# B&R Automation Studio project acopos6d_issues (part 5)

#### FastLib.fun - Exported functions and function blocks
```iecst
FUNCTION_BLOCK fdStationQueueControl
	VAR_INPUT
		Enable : BOOL;
		ReleaseShuttles : BOOL;
		ShuttleList : ARRAY[0..fdSTATION_SHUTTLE_LAST_INDEX] OF MpTrafficShuttleInfoType;
		ShuttleCapacity : UINT; (*Count how many shuttles process station can handle*)
		pStation : REFERENCE TO MpTrafficStationControl;
	END_VAR
	VAR_OUTPUT
		ShuttleReleaseDone : BOOL;
		ShuttleReleaseAborted : BOOL;
		ReleaseShuttle : BOOL;
		NumOccypyingShuttles : UINT;
	END_VAR
	VAR
		state : DINT;
		lastState : DINT;
		loop : DINT;
		index : DINT;
		shuttleFound : BOOL;
		shuttleIDToRelease : UINT;
		shuttleIDToAutoRelease : UINT;
	END_VAR
END_FUNCTION_BLOCK

FUNCTION_BLOCK fdTiltAround
	VAR_INPUT
		Execute : {REDUND_UNREPLICABLE} BOOL;
		MaxAngle : {REDUND_UNREPLICABLE} REAL;
		Steps : {REDUND_UNREPLICABLE} DINT;
		Velocity : McAcp6DShortAxAxesType;
		Shuttle : REFERENCE TO Mc6DShuttleType;
	END_VAR
	VAR_OUTPUT
		Acknowledge : BOOL;
		Error : BOOL;
	END_VAR
	VAR
		state : DINT;
		step : DINT;
		MoveShortAxis : MC_BR_MoveShortAxis_Acp6D;
	END_VAR
END_FUNCTION_BLOCK

FUNCTION_BLOCK fdWaitUntilAllDone
	VAR_INPUT
		Execute : {REDUND_UNREPLICABLE} BOOL;
		Shuttles : {REDUND_UNREPLICABLE} ARRAY[0..fdMAX_WAIT_SHUTTLE_COUNT] OF Mc6DShuttleType;
	END_VAR
	VAR_OUTPUT
		Done : BOOL;
		Error : BOOL;
		WaitingFor : UINT;
	END_VAR
	VAR
		state : DINT;
		i : DINT;
		ShGetInfo : MC_BR_ShGetInfo_Acp6D;
	END_VAR
END_FUNCTION_BLOCK

FUNCTION_BLOCK fdPulse
	VAR_INPUT
		Execute : {REDUND_UNREPLICABLE} BOOL;
		T_on : {REDUND_UNREPLICABLE} TIME;
		T_off : {REDUND_UNREPLICABLE} TIME;
	END_VAR
	VAR_OUTPUT
		Q : BOOL;
	END_VAR
	VAR
		state : DINT;
		TON_on : TON;
		TON_off : TON;
	END_VAR
END_FUNCTION_BLOCK

FUNCTION_BLOCK fdFindZone
	VAR_INPUT
		Assembly : REFERENCE TO Mc6DAssemblyType; (*The assembly reference establishes the connection between the function block and the assembly.*)
		Execute : BOOL;
		Name : STRING[32];
	END_VAR
	VAR_OUTPUT
		ZoneFound : BOOL;
		ZoneNotFound : BOOL;
		Error : BOOL;
		Zone : Mc6DZoneType; (* Zone reference *)
		ZoneInfo : McAcp6DGetZoneAddInfoType;
	END_VAR
	VAR
		state : DINT;
		i : DINT;
		AsmGetZone : MC_BR_AsmGetZone_Acp6D;
		lastZoneID : UINT;
	END_VAR
END_FUNCTION_BLOCK

FUNCTION_BLOCK fdStation
	VAR_INPUT
		Assembly : REFERENCE TO Mc6DAssemblyType;
		TrafficManager : REFERENCE TO MpTrafficManagerType;
		Station : REFERENCE TO MpTrafficStationType;
		NextStation : REFERENCE TO MpTrafficStationType;
		Enable : BOOL;
		NextState : BOOL;
		JumpToState : UINT;
		Parameters : fdStationParametersType;
		Commands : fdStationCommandsType;
		Operation : fdStationOperationType;
		Loop : DINT;
		StateInfo : STRING[80];
	END_VAR
	VAR_OUTPUT
		State : UINT;
		Active : BOOL;
		NumOccupyingShuttles : UINT;
		CommandDone : BOOL;
		CommandAcknowledge : BOOL;
		CommandError : BOOL;
		ErrorID : DINT;
		ErroredSequenceState : DINT;
		Shuttles : fdStationShuttlesType;
		VirtualShuttle : MpTrafficShuttleInfoType;
		MacroShuttle : MpTrafficShuttleInfoType;
	END_VAR
	VAR
		m_sequence_state : DINT;
		m_control : fdStationMemberControlType;
		m_move : fdStationMemberMoveType;
		m_group : fdStationMemberGroupType;
		m_macro : fdStationMemberMacroType;
		m_zone : fdStationMemberZoneType;
		m_cmd : fdStationMemberCommandType;
		m_status : fdStationMemberStatusType;
		m_var : fdStationMemberVarType;
	END_VAR
END_FUNCTION_BLOCK
(**)

FUNCTION_BLOCK fdMove6DSync
	VAR_INPUT
		Shuttle : REFERENCE TO Mc6DShuttleType;
		Execute : BOOL;
		Home : BOOL;
		Parameters : fdMove6DSyncParametersType;
	END_VAR
	VAR_OUTPUT
		Acknowledge : BOOL;
		Done : BOOL;
		Error : BOOL;
		ErrorID : DINT;
		CurrentPosition : McAcp6DShPositionType;
	END_VAR
	VAR
		state : DINT;
		i : DINT;
		ShGetInfo : MC_BR_ShGetInfo_Acp6D;
		Move6D : MC_BR_Move6D_Acp6D;
		m : fdMove6DSyncMemberType;
	END_VAR
END_FUNCTION_BLOCK

FUNCTION fdCalcTimeToTarget : REAL
	VAR_INPUT
		Distance : REAL;
		MaxVelocity : REAL;
		Acceleration : REAL;
	END_VAR
	VAR
		timeToMaxVelocity : REAL;
		distanceToMaxVelocity : REAL;
		distanceToTarget : REAL;
	END_VAR
END_FUNCTION

FUNCTION fdCalcTargetVelocity : REAL
	VAR_INPUT
		Distance : REAL;
		TimeToTarget : REAL;
		Acceleration : REAL;
	END_VAR
	VAR
		minimumVelocity : REAL;
		discriminant : REAL;
		a : REAL;
		b : REAL;
		c : REAL;
		x1 : REAL;
		x2 : REAL;
	END_VAR
END_FUNCTION
```

#### fdStationQueueControl.st
```iecst
(*  *)
FUNCTION_BLOCK fdStationQueueControl

	IF NOT Enable THEN
		state := 0;
		ReleaseShuttle := FALSE;
		ShuttleReleaseDone := FALSE;
		ShuttleReleaseAborted := FALSE;
	END_IF;

	CASE state OF
		0:
			// -----------------------------------------------------------------
			IF ReleaseShuttles THEN
				IF pStation.Info.NumOccupyingShuttles > 0 THEN
					index := 0;
					state := 100;
				ELSE
					state := 199;
				END_IF;
			ELSIF pStation.Info.NumOccupyingShuttles > ShuttleCapacity THEN
				shuttleIDToAutoRelease := pStation.Info.LastArrivedShuttle.ShuttleID;
				// Station is executing current process and there is no room for more shuttles ->
				// release queuing extra shuttles straight forward
				loop := 0;
				state := 200;
			END_IF;

		100:
			// Manual queue release sequence
			// ----------------------------------------------------------------------------------------------------------------------------------
			// Select the next requested shuttle from the shuttle list
			shuttleFound := FALSE;

			WHILE index <= fdSTATION_SHUTTLE_LAST_INDEX DO
				IF ShuttleList[index].ShuttleID > 0 THEN
					shuttleIDToRelease := ShuttleList[index].ShuttleID;
					shuttleFound := TRUE;
					index := index + 1;
					EXIT;
				END_IF;
				index := index + 1;
			END_WHILE;

			IF shuttleFound THEN
				// Proceed to release next shuttle
				loop := 0;
				state := 110;
			ELSE
				// No more shuttles to release
				state := 199;
			END_IF;
		110:
			// Select shuttle to be released from stations shuttle list
			// -----------------------------------------------------------------
			IF loop > pStation.Info.NumOccupyingShuttles THEN
				// whole list has been checked through and we cant find requested shuttle -> move on
				state := 100;
			ELSIF pStation.SelectedShuttle.ShuttleID = shuttleIDToRelease THEN
				state := 130;
			ELSE
				loop := loop  + 1;
				pStation(SelectNextShuttle := TRUE);
				pStation(SelectNextShuttle := FALSE);
			END_IF;
		130:
			// Release the shuttle
			// -----------------------------------------------------------------
			ReleaseShuttle := TRUE;

			IF pStation.ReleaseDone THEN
				state := 100;
			ELSIF pStation.ReleaseAborted THEN
				state := 300;
			END_IF;
		199:
			// Done
			// -----------------------------------------------------------------
			ShuttleReleaseDone := TRUE;

			IF NOT ReleaseShuttles THEN
				state := 0;
			END_IF;

		200:
			// Automatic queue release sequence
			// ----------------------------------------------------------------------------------------------------------------------------------
			// Select shuttle to be released from stations shuttle list
			// -----------------------------------------------------------------
			IF loop > pStation.Info.NumOccupyingShuttles THEN
				// whole list has been checked through and we cant find requested shuttle -> move on
				state := 0;
			ELSIF pStation.SelectedShuttle.ShuttleID = shuttleIDToAutoRelease THEN
				state := 210;
			ELSE
				loop := loop  + 1;
				pStation(SelectNextShuttle := TRUE);
				pStation(SelectNextShuttle := FALSE);
			END_IF;
		210:
			// Release the queuing shuttle
			// -----------------------------------------------------------------
			ReleaseShuttle := TRUE;

			IF pStation.ReleaseDone THEN
				state := 0;
			ELSIF pStation.ReleaseAborted THEN
				state := 300;
			END_IF;

		300:
			// Error
			// -----------------------------------------------------------------
			ShuttleReleaseAborted := TRUE;

	END_CASE;

	IF state <> lastState THEN
		lastState := state;
		ReleaseShuttle := FALSE;
		ShuttleReleaseDone := FALSE;
		ShuttleReleaseAborted := FALSE;
	END_IF;

	NumOccypyingShuttles := pStation.Info.NumOccupyingShuttles;

END_FUNCTION_BLOCK
```

#### fdTiltAround.st
```iecst
(*  *)
FUNCTION_BLOCK fdTiltAround

	IF NOT Execute THEN
		MoveShortAxis.Execute := FALSE;
		step := 0;
		state := 0;
	END_IF;

	CASE state OF
		0:
			IF Execute THEN
				state := 10;
			END_IF;
		10:
			IF step > Steps THEN
				state := 100;
			ELSE
				MoveShortAxis.Parameters.Position.Rx := MaxAngle * SIN((2 * brmPI / Steps) * step);
				MoveShortAxis.Parameters.Position.Ry := MaxAngle * COS((2 * brmPI / Steps) * step);
				MoveShortAxis.Parameters.Position.Rz := 0;
				MoveShortAxis.Parameters.Position.Z := 0.004;
				state := 20;
			END_IF;
		20:
			MoveShortAxis.Execute := TRUE;

			IF MoveShortAxis.Acknowledge THEN
				MoveShortAxis.Execute := FALSE;
				step := step + 1;
				state := 10;
			END_IF;
		100:
//			MoveShortAxis.Parameters.Position.Rx := 0;
//			MoveShortAxis.Parameters.Position.Ry := 0;
//			MoveShortAxis.Parameters.Position.Rz := 0;
//			MoveShortAxis.Parameters.Position.Z := 0.001;
//			MoveShortAxis.Execute := TRUE;
//
//			IF MoveShortAxis.Done OR MoveShortAxis.Acknowledge THEN
//				MoveShortAxis.Execute := FALSE;
//				step := step + 1;
//				state := 101;
//			END_IF;

			IF NOT Execute THEN
				state := 0;
			END_IF;
	END_CASE;

	MoveShortAxis.Shuttle := ADR(Shuttle);
	MoveShortAxis.Parameters.Mode :=  mcACP6D_MOVE_ABSOLUTE;
	MoveShortAxis.Parameters.Velocity := Velocity;
	MoveShortAxis();

	Acknowledge := (state = 100);
	Error := MoveShortAxis.Error;

END_FUNCTION_BLOCK
```

#### fdWaitUntilIdle.st
```iecst
(*  *)
FUNCTION_BLOCK fdWaitUntilAllDone

	IF NOT Execute THEN
		state := 0;
		i := 0;
		ShGetInfo.Execute := FALSE;
		WaitingFor := 0;
	END_IF;

	CASE state OF
		0:
			IF Execute THEN
				state := 10;
			END_IF;
		10:
			IF i > fdMAX_STATION_SHUTTLE_COUNT THEN
				state := 100;
			ELSE
				IF Shuttles[i].controlif = 0 THEN
					// Not a valid shuttle reference. Move to next item in the list
					i := i + 1;
				ELSE
					state := 20;
				END_IF;
			END_IF;
		20:
			ShGetInfo.Execute := TRUE;

			IF ShGetInfo.Done THEN
				WaitingFor := ShGetInfo.ShuttleInfo.ShuttleID;

				IF (ShGetInfo.ShuttleInfo.State =  mcACP6D_SH_STATE_IDLING) AND (ShGetInfo.ShuttleInfo.MotionBuffer.NumberOfCommands = 0) THEN
					i := i + 1;
					state := 10;
				END_IF;
				ShGetInfo.Execute := FALSE;

			ELSIF ShGetInfo.Error THEN
				ShGetInfo.Execute := FALSE;
				state := 101;
			END_IF;
		100:
			IF NOT Execute THEN
				state := 0;
			END_IF;
	END_CASE;

	ShGetInfo.Shuttle := ADR(Shuttles[i]);
	ShGetInfo();

	Done := (state = 100);
	Error := ShGetInfo.Error;

END_FUNCTION_BLOCK
```

#### fdPulse.st
```iecst
(*  *)
FUNCTION_BLOCK fdPulse

	IF NOT Execute THEN
		state := 0;
	END_IF;

	CASE state OF
		0:
			IF Execute THEN
				state := 10;
			END_IF;
		10:
			IF TON_on.Q THEN
	  			state := 20;
			END_IF;
		20:
			IF TON_off.Q THEN
				state := 10;
			END_IF;
		100:
			IF NOT Execute THEN
				state := 0;
			END_IF;
	END_CASE;

	TON_on.IN := (state = 10);
	TON_on.PT := T_on;
	TON_on();

	TON_off.IN := (state = 20);
	TON_off.PT := T_off;
	TON_off();

	Q := (state = 10);

END_FUNCTION_BLOCK
```

#### fdFindZone.st
```iecst
(*  *)
FUNCTION_BLOCK fdFindZone

	IF NOT Execute THEN
		state := 0;
		i := 0;
		AsmGetZone.Enable := FALSE;
		ZoneFound := FALSE;
		ZoneNotFound := FALSE;
		Error := FALSE;
		brsmemset(ADR(ZoneInfo), 0, SIZEOF(ZoneInfo));
		brsmemset(ADR(Zone), 0, SIZEOF(Zone));
	END_IF;

	CASE state OF
		0:
			// --------------------------------------------
			IF Execute THEN
				state := 10;
			END_IF;
		10:
			// --------------------------------------------
			AsmGetZone.Enable := TRUE;
			IF AsmGetZone.Valid THEN
				IF AsmGetZone.TotalCount = 0 THEN
					state := 101;
				ELSE
					state := 20;
				END_IF;
			END_IF;
		20:
			// --------------------------------------------
			lastZoneID := AsmGetZone.AdditionalInfo.ZoneID;

			IF brsmemcmp(ADR(AsmGetZone.AdditionalInfo.Name), ADR(Name), SIZEOF(Name)) = 0 THEN
				// Names match -> found
				Zone := AsmGetZone.Zone;
				ZoneInfo := AsmGetZone.AdditionalInfo;
				state := 100;
			ELSE
				IF AsmGetZone.RemainingCount = 0 THEN
					state := 101;
				ELSE
					state := 30;
				END_IF;
			END_IF;
		30:
			// --------------------------------------------
			IF AsmGetZone.AdditionalInfo.ZoneID <> lastZoneID THEN
				state := 20;
			END_IF;

		100:
			// --------------------------------------------
			ZoneFound := TRUE;
		101:
			// --------------------------------------------
			ZoneNotFound := TRUE;
		102:
			// --------------------------------------------
			Error := TRUE;
	END_CASE;

	AsmGetZone.Assembly := ADR(Assembly);
	AsmGetZone.Next := (state = 30);
	AsmGetZone();

END_FUNCTION_BLOCK
```

#### fdMove6DSync.st
```iecst
//
FUNCTION fdCalcTimeToTarget

	// v = a * t -> t = v / a
	timeToMaxVelocity := MaxVelocity / Acceleration;

	// Displacement: s = v_0 * t + 0.5 * at^2 -> s = 0.5 * at^2
	distanceToMaxVelocity := 0.5 * Acceleration * brmpow(timeToMaxVelocity, 2);

	// Displacement: s = v_0 * t + 0.5 * at^2 -> t = sqrt((2s)/a)
	IF distanceToMaxVelocity > Distance THEN
		// Case where we never hit the target velocity
		fdCalcTimeToTarget := SQRT(2 * Distance / Acceleration);
	ELSE
		// Case where we reach target velocity
		distanceToTarget := Distance - distanceToMaxVelocity;

		fdCalcTimeToTarget := SQRT(2 * distanceToMaxVelocity / Acceleration) + distanceToTarget / MaxVelocity;
	END_IF;

END_FUNCTION

//
FUNCTION fdCalcTargetVelocity

	// This seems to be rougly minimum velocity 6D system can do
	minimumVelocity := 0.0001;

	IF Distance < 0.001 THEN
		fdCalcTargetVelocity := minimumVelocity;
	END_IF;

	// Move consists of two parts, 1st is acceleration to end velocity and 2nd is constant velocity part
	// We know following:
	// TimeToTarget = t1 + t2
	// TargetVelocity = Acceleration * t1
	// s2 = TargetVelocity * t2
	// Distance = s1 + s2
	// s1 = 0.5 * Acceleration * t1^2

	// Solve with quadratic equation
	// x = (-b +- SQRT((b^2)-4ac))/2a
	// discriminant = b*b - 4*a*c;
	a := 0.5;
	b := -1 * TimeToTarget * Acceleration;
	c := Acceleration * Distance;

	// Solve discriminant for the equation
	discriminant := b * b - 4 * a * c;

	IF (discriminant > 0) THEN
		// Two real and distinct roots
		x1 := (-1 * b + SQRT(discriminant)) / (2*a);
		x2 := (-1 * b - SQRT(discriminant)) / (2*a);

		IF x1 >= 0 AND x2 >= 0 THEN
			fdCalcTargetVelocity := MIN(x1, x2);
		ELSIF x1 > 0 THEN
			fdCalcTargetVelocity := x1;
		ELSIF x2 > 0 THEN
			fdCalcTargetVelocity := x2;
		ELSE
			// Both are negative -> impossible situation as velocity cant be negative in this case
			fdCalcTargetVelocity := 0;
		END_IF;

	ELSIF (discriminant = 0) THEN
		// One real root (repeated)
		fdCalcTargetVelocity := -1 * b / (2*a);
	ELSE
		// No real solution -> set to zero so it errors out as this is impossible request
		fdCalcTargetVelocity := 0;
	END_IF

	//fdCalcTargetVelocity := MAX(MinimumVelocity, fdCalcTargetVelocity);

END_FUNCTION

(*  *)
FUNCTION_BLOCK fdMove6DSync

	CASE state OF
		0:
			// --------------------------------------------
			ShGetInfo.Execute := FALSE;
			Move6D.Execute := FALSE;
			ErrorID := 0;
			m.PositionUpdatePending := FALSE;

			IF Execute THEN
				state := 100;
			ELSIF Home THEN
				state := 200;
			END_IF;

		100:
			// Calculate target velocities for all axis
			// --------------------------------------------
			// Calculate distance each axis needs to travel
			m.DistanceToTarget.InPlane := SQRT(brmpow(Parameters.Position.X - CurrentPosition.X, 2) + brmpow(Parameters.Position.Y - CurrentPosition.Y, 2));
			m.DistanceToTarget.Z := ABS(Parameters.Position.Z - CurrentPosition.Z);
			m.DistanceToTarget.Rx := ABS(Parameters.Position.Rx - CurrentPosition.Rx);
			m.DistanceToTarget.Ry := ABS(Parameters.Position.Ry - CurrentPosition.Ry);
			m.DistanceToTarget.Rz := ABS(Parameters.Position.Rz - CurrentPosition.Rz);

			// Calculate which axis takes longest to reach its target from current position
			m.TimeToTarget.InPlane := fdCalcTimeToTarget(m.DistanceToTarget.InPlane, Parameters.Velocity.InPlane, Parameters.Acceleration.InPlane);
			m.TimeToTarget.Z := fdCalcTimeToTarget(m.DistanceToTarget.Z, Parameters.Velocity.Z, Parameters.Acceleration.Z);
			m.TimeToTarget.Rx := fdCalcTimeToTarget(m.DistanceToTarget.Rx, Parameters.Velocity.Rx, Parameters.Acceleration.Rx);
			m.TimeToTarget.Ry := fdCalcTimeToTarget(m.DistanceToTarget.Ry, Parameters.Velocity.Ry, Parameters.Acceleration.Ry);
			m.TimeToTarget.Rz := fdCalcTimeToTarget(m.DistanceToTarget.Rz, Parameters.Velocity.Rz, Parameters.Acceleration.Rz);

			// The axis that takes the longest to reach the target
			m.LongestTimeToTarget := MAX(m.TimeToTarget.InPlane, m.TimeToTarget.Z, m.TimeToTarget.Rx, m.TimeToTarget.Ry, m.TimeToTarget.Rz);

			m.TargetVelocity.InPlane := fdCalcTargetVelocity(m.DistanceToTarget.InPlane, m.LongestTimeToTarget, Parameters.Acceleration.InPlane);
			m.TargetVelocity.Z := fdCalcTargetVelocity(m.DistanceToTarget.Z, m.LongestTimeToTarget, Parameters.Acceleration.Z);
			m.TargetVelocity.Rx := fdCalcTargetVelocity(m.DistanceToTarget.Rx, m.LongestTimeToTarget, Parameters.Acceleration.Rx);
			m.TargetVelocity.Ry := fdCalcTargetVelocity(m.DistanceToTarget.Ry, m.LongestTimeToTarget, Parameters.Acceleration.Ry);
			m.TargetVelocity.Rz := fdCalcTargetVelocity(m.DistanceToTarget.Rz, m.LongestTimeToTarget, Parameters.Acceleration.Rz);

			state := 101;
		101:
			// Execute the move
			// -------------------------------------------
			Move6D.Parameters.InPlane.Acceleration := Parameters.Acceleration.InPlane;
			Move6D.Parameters.InPlane.Velocity := m.TargetVelocity.InPlane;
			Move6D.Parameters.InPlane.Position.X := Parameters.Position.X;
			Move6D.Parameters.InPlane.Position.Y := Parameters.Position.Y;

			Move6D.Parameters.ShortAxis.Velocity.Z := m.TargetVelocity.Z;
			Move6D.Parameters.ShortAxis.Velocity.Rx := m.TargetVelocity.Rx;
			Move6D.Parameters.ShortAxis.Velocity.Ry := m.TargetVelocity.Ry;
			Move6D.Parameters.ShortAxis.Velocity.Rz := m.TargetVelocity.Rz;
			Move6D.Parameters.ShortAxis.Position.Z := Parameters.Position.Z;
			Move6D.Parameters.ShortAxis.Position.Rx := Parameters.Position.Rx;
			Move6D.Parameters.ShortAxis.Position.Ry := Parameters.Position.Ry;
			Move6D.Parameters.ShortAxis.Position.Rz := Parameters.Position.Rz;
			Move6D.Execute := TRUE;

			IF Move6D.Done OR Move6D.Acknowledge THEN
	  			m.PositionUpdatePending := TRUE;
			END_IF;

			IF NOT Execute THEN
				IF m.PositionUpdatePending THEN
					m.PositionUpdatePending := FALSE;
	  				CurrentPosition := Parameters.Position;
				END_IF;
				Move6D.Execute := FALSE;
				state := 0;
			END_IF;

		200:
			// Home shuttle by reading its current location
			// --------------------------------------------
			ShGetInfo.Execute := TRUE;

			IF NOT Home THEN
				ShGetInfo.Execute := FALSE;
				state := 0;
			ELSIF ShGetInfo.Done THEN
				CurrentPosition := ShGetInfo.ShuttleInfo.Position;
			ELSIF ShGetInfo.Error THEN
				ErrorID := ShGetInfo.ErrorID;
			END_IF;
	END_CASE;

	// Functions
	// --------------------------------------------
	ShGetInfo.Shuttle := ADR(Shuttle);
	ShGetInfo();

	Move6D.Shuttle := ADR(Shuttle);
	Move6D();

	// --------------------------------------------
	Done := Move6D.Done OR ShGetInfo.Done;
	Acknowledge := Move6D.Acknowledge;
	Error := Move6D.Error OR ShGetInfo.Done;

END_FUNCTION_BLOCK
```

#### fdStation.st
```iecst
(* *)
FUNCTION_BLOCK fdStation

	// Station enable control
	// ----------------------------------------------------------------------------------------
	m_control.Enable_EdgeNegative(CLK := Enable);

	IF m_control.Enable_EdgeNegative.Q THEN
		IF Active THEN
			// Jump to
	  		m_sequence_state := 90;
		ELSE
			m_sequence_state := 0;
		END_IF;
	END_IF;

	// External state control
	// ----------------------------------------------------------------------------------------
	IF Active THEN
		IF NextState THEN
			State := State + 1;
			m_var.StateChanged := TRUE;
		ELSIF JumpToState <> State THEN
			State := JumpToState;
			m_var.StateChanged := TRUE;
		END_IF;

		IF m_var.StateChanged THEN
			m_var.StateChanged := FALSE;
			NextState := FALSE;
			JumpToState := State;;
			brsmemset(ADR(Commands), 0, SIZEOF(Commands));
			JumpToState := State;;
		END_IF;
	END_IF;

	// Check if all commands are reset
	// -----------------------------------------------------------------
	m_var.NoCommandActive := (brsmemcmp(ADR(m_var.NoCommands), ADR(Commands), SIZEOF(Commands)) = 0);

	// Station command sequence
	// -----------------------------------------------------------------
	CASE m_sequence_state OF
		0:
			StateInfo := 'Station disabled';
			// -----------------------------------------------------------------
			Active := FALSE;
			State := 0;
			NextState := FALSE;
			JumpToState := 0;
			Loop := 0;
			brsmemset(ADR(Commands), 0, SIZEOF(Commands));
			brsmemset(ADR(Operation), 0, SIZEOF(Operation));
			brsmemset(ADR(m_var), 0, SIZEOF(m_var));
			brsmemset(ADR(m_cmd), 0, SIZEOF(m_cmd));
			brsmemset(ADR(m_status), 0, SIZEOF(m_status));

			IF Enable THEN
	  			m_sequence_state := m_sequence_state + 1;
			END_IF;
		1:
			StateInfo := 'Wait for station to be active and open';
			// -----------------------------------------------------------------
			IF m_control.StationControl.Active AND m_control.StationControl.State = mpTRAFFIC_ST_ON_OPEN THEN
				m_sequence_state := m_sequence_state + 1;
			END_IF
		2:
			StateInfo := 'Create shuttle group';
			// -----------------------------------------------------------------
			m_cmd.GroupCreate := TRUE;
			IF m_group.Create.Done THEN
				m_var.ShuttleGroup := m_group.Create.ShuttleGroup;
				m_sequence_state := 10;
			ELSIF m_group.Create.Error THEN
				m_status.ErrorID := m_group.Create.ErrorID;
			END_IF;
		10:
			StateInfo := 'Check if virtual shuttle exists';
			// -----------------------------------------------------------------
			IF NOT Parameters.CreateVirtualShuttle THEN
				// Virtual shuttle not needed in this station -> move on
				brsmemset(ADR(VirtualShuttle), 0, SIZEOF(VirtualShuttle));
				m_sequence_state := 20;
			ELSE
				IF VirtualShuttle.Shuttle6D.controlif = 0 THEN
					// Virtual shuttle does not exist -> create new one
					m_sequence_state := m_sequence_state + 1;
				ELSE
					// Virtual shuttle already exists in this station -> read its information
					m_sequence_state := 12;
				END_IF;
			END_IF;
		11:
			StateInfo := 'Create virtual shuttle';
			// -----------------------------------------------------------------
			m_cmd.VirtualShuttleCreate := TRUE;

			IF m_control.VirtualShuttleCreate.Done THEN
				VirtualShuttle.Shuttle6D := m_control.VirtualShuttleCreate.VirtualShuttle;
				m_sequence_state := m_sequence_state + 1;
			ELSIF m_control.VirtualShuttleCreate.Error THEN
				m_status.ErrorID := m_control.VirtualShuttleCreate.ErrorID;
			END_IF;
		12:
			StateInfo := 'Read virtual shuttle ID';
			// -----------------------------------------------------------------
			m_control.GetShuttleInfo.Shuttle := ADR(VirtualShuttle.Shuttle6D);
			m_cmd.GetShuttleInfo := TRUE;

			IF m_control.GetShuttleInfo.Done THEN
				VirtualShuttle.ShuttleID := m_control.GetShuttleInfo.ShuttleInfo.ShuttleID;
				m_sequence_state := 20;
			ELSIF m_control.GetShuttleInfo.Error THEN
				m_status.ErrorID := m_control.GetShuttleInfo.ErrorID;
			END_IF;

		20:
			StateInfo := 'Find station zone by name';
			// -----------------------------------------------------------------
			IF brsstrlen(ADR(Parameters.Zone.Name)) = 0 THEN
				m_var.str := DINT_TO_STRING(Parameters.StationNumber);
				Parameters.Zone.Name := CONCAT('Zone', m_var.str);
			END_IF;

			brsmemset(ADR(m_zone.Zone), 0, SIZEOF(m_zone.Zone));
			m_zone.Find.Name := Parameters.Zone.Name;
			m_cmd.ZoneFind := TRUE;

			IF m_zone.Find.ZoneFound THEN
				m_zone.Zone := m_zone.Find.Zone;
				m_sequence_state := 30;
			ELSIF m_zone.Find.ZoneNotFound THEN
				m_sequence_state := m_sequence_state + 1;
			END_IF;
		21:
			StateInfo := 'Create zone';
			// -----------------------------------------------------------------
			m_zone.Create.Parameters.BottomLeft := Parameters.Zone.BottomLeft;
			m_zone.Create.Parameters.TopRight := Parameters.Zone.TopRight;
			m_zone.Create.Parameters.Name := Parameters.Zone.Name;
			m_cmd.ZoneCreate := TRUE;

			IF m_zone.Create.Done THEN
				// Go back one step and rescan the zones to get the zone reference
				m_sequence_state := 20;
			ELSIF m_zone.Create.Error THEN
				m_status.ErrorID := m_zone.Create.ErrorID;
			END_IF;

		30:
			StateInfo := 'Delete old macro if it exists';
			// -----------------------------------------------------------------
			IF brsstrlen(ADR(Parameters.MacroName)) = 0 THEN
				m_var.str := DINT_TO_STRING(Parameters.StationNumber);
				Parameters.MacroName := CONCAT('Macro', m_var.str);
			END_IF;

			m_macro.Delete.Name := Parameters.MacroName;
			m_cmd.MacroDelete := TRUE;

			// Move forward if "macro name not defined" error is received
			IF (m_macro.Delete.Done) OR (m_macro.Delete.Error AND m_macro.Delete.ErrorID = - 1065811714) THEN
				m_sequence_state := m_sequence_state + 1;
			ELSIF m_macro.Delete.Error THEN
				m_status.ErrorID := m_macro.Delete.ErrorID;
			END_IF;
		31:
			StateInfo := 'Create new macro';
			// -----------------------------------------------------------------
			m_macro.Create.Parameters.Name := Parameters.MacroName;
			m_cmd.MacroCreate := TRUE;

			IF m_macro.Create.Done THEN
				m_var.MacroShuttle.Shuttle6D := m_macro.Create.MacroShuttle;
				m_sequence_state := 100;
			ELSIF m_macro.Create.Error THEN
				m_status.ErrorID := m_macro.Create.ErrorID;
			END_IF;

		90:
			StateInfo := 'Deactivating - Clear group';
			// -----------------------------------------------------------------
			m_cmd.GroupClear := TRUE;
			IF m_group.Clear.Done THEN
	  			m_sequence_state := m_sequence_state + 1;
			END_IF;
		91:
			StateInfo := 'Deactivating - Delete group';
			// -----------------------------------------------------------------
			m_cmd.GroupDelete := TRUE;
			IF m_group.Delete.Done THEN
				m_sequence_state := m_sequence_state + 1;
			END_IF;
		92:
			StateInfo := 'Deactivating - Decouple planet system';
			// -----------------------------------------------------------------
			FOR m_var.index := 0 TO fdSTATION_SHUTTLE_LAST_INDEX DO
				m_move.SunPlanet.Parameters.ShuttleList[m_var.index].Shuttle := ADR(m_var.Shuttles.List[m_var.index].Shuttle6D);
			END_FOR;

			m_move.SunPlanet.Parameters.Option := mcACP6D_PLANET_REMOVE_SH;
			m_cmd.Input.SunPlanet.Decouple := TRUE;

			IF m_move.SunPlanet.Done OR (m_move.SunPlanet.ErrorID = -1065795584) THEN
				// Error -1065795584 indicates invalid parameters. A generic issue if shuttles are not currently
				// grouped around sun shuttle. -> just move on
	  			m_sequence_state := m_sequence_state + 1;
			END_IF;
		93:
			StateInfo := 'Deactivating - Delete macro';
			// -----------------------------------------------------------------
			m_cmd.MacroDelete := TRUE;
			IF m_macro.Delete.Done THEN
				m_sequence_state := 99;
			END_IF;
		99:
			StateInfo := 'Deactivating - Deactivation complete';
			// -----------------------------------------------------------------
			m_sequence_state := 0;

		100:
			// Waiting for commands
			// -----------------------------------------------------------------
			Active := TRUE;

			IF Commands.AddShuttle THEN
				m_sequence_state := 110;
			ELSIF Commands.ReleaseAllShuttles THEN
				m_sequence_state := 120;
			ELSIF Commands.MacroRun THEN
				m_sequence_state := 130;
			ELSIF Commands.MacroSave THEN
				m_sequence_state := 140;
			ELSIF Commands.MoveInPlane THEN
				m_sequence_state := 150;
			ELSIF Commands.MoveArc THEN
				m_sequence_state := 160;
			ELSIF Commands.MoveShortAxis THEN
				m_sequence_state := 170;
			ELSIF Commands.Move6D THEN
				m_sequence_state := 180;
			ELSIF Commands.Spin THEN
				m_sequence_state := 190;
			ELSIF Commands.WaitCommandLabel THEN
				m_sequence_state := 200;
			ELSIF Commands.WaitUntilAllDone THEN
				m_sequence_state := 210;
			ELSIF Commands.Group.Couple_CommonCenterPoint THEN
				m_sequence_state := 220;
			ELSIF Commands.Group.Couple_OwnCenterPoint THEN
				m_sequence_state := 221;
			ELSIF Commands.Group.Decouple THEN
				m_sequence_state := 230;
			ELSIF Commands.SunPlanet.Couple THEN
				m_sequence_state := 240;
			ELSIF Commands.SunPlanet.Decouple THEN
				m_sequence_state := 250;
			END_IF;

		110:
			// Add new shuttle to station if there is room for it
			// -----------------------------------------------------------------
			IF m_var.NoCommandActive THEN
				m_sequence_state := 100;
			ELSIF m_var.Shuttles.Count <= fdSTATION_SHUTTLE_LAST_INDEX THEN
				m_var.Shuttles.List[m_var.Shuttles.Count] := m_control.StationControl.Info.LastArrivedShuttle;
				m_var.Shuttles.Count := m_var.Shuttles.Count + 1;
				m_sequence_state := m_sequence_state + 1;
			ELSE
				m_status.CommandError := TRUE;
				m_status.ErrorID := m_sequence_state;
			END_IF;

		111:
			// Clear group before adding ALL shuttles as we cant add one by one
			// -----------------------------------------------------------------
			m_cmd.GroupClear := TRUE;

			m_status.CommandError := m_group.Clear.Error;
			m_status.ErrorID := m_group.Clear.ErrorID;

			IF m_var.NoCommandActive THEN
				m_sequence_state := 100;
			ELSIF m_group.Clear.Done THEN
				m_sequence_state := m_sequence_state + 1;
			END_IF;
		112:
			// Add shuttles to shuttle group
			// -----------------------------------------------------------------
			brsmemset(ADR(m_group.AddShuttle.Parameters.ShuttleList), 0, SIZEOF(m_group.AddShuttle.Parameters.ShuttleList));

			FOR m_var.index := 0 TO m_var.Shuttles.Count - 1 DO
				m_group.AddShuttle.Parameters.ShuttleList[m_var.index].Shuttle := ADR(m_var.Shuttles.List[m_var.index].Shuttle6D);
			END_FOR;

			m_cmd.GroupAddShuttle := TRUE;

			m_status.CommandDone := m_group.AddShuttle.Done;
			m_status.CommandError := m_group.AddShuttle.Error;
			m_status.ErrorID := m_group.AddShuttle.ErrorID;

			IF m_var.NoCommandActive THEN
				m_sequence_state := 100;
			END_IF;

		120:
			// Clear group
			// -----------------------------------------------------------------
			m_cmd.GroupClear := TRUE;

			m_status.CommandError := m_group.Clear.Error;
			m_status.ErrorID := m_group.Clear.ErrorID;

			IF m_var.NoCommandActive THEN
				m_sequence_state := 100;
			ELSIF m_group.Clear.Done THEN
				m_sequence_state := m_sequence_state + 1;
			END_IF;

		121:
			// Release shuttles from station
			// -----------------------------------------------------------------
			m_cmd.Input.ReleaseAllShuttles := TRUE;

			m_status.CommandError := m_control.StationQueueControl.ShuttleReleaseAborted;
			m_status.ErrorID := m_sequence_state;

			IF m_var.NoCommandActive THEN
				m_sequence_state := 100;
			ELSIF m_control.StationQueueControl.ShuttleReleaseDone THEN
				m_sequence_state := m_sequence_state + 1;
			END_IF;

		122:
			// Wait until shuttles have left the station
			// -----------------------------------------------------------------
			m_cmd.ZoneGetBarrierInfo := TRUE;

			m_status.CommandError := m_zone.GetBarrierInfo.Error;
			m_status.ErrorID := m_zone.GetBarrierInfo.ErrorID;

			IF m_var.NoCommandActive THEN
				m_sequence_state := 100;
			ELSIF m_zone.GetBarrierInfo.Done THEN
				m_cmd.ZoneGetBarrierInfo := FALSE;
				IF m_zone.GetBarrierInfo.BarrierInfo.NumberOfShuttles = 0 THEN
					m_var.Shuttles.Count := 0;
					brsmemset(ADR(m_var.Shuttles.List), 0, SIZEOF(m_var.Shuttles.List));
					m_status.CommandDone := TRUE;
				END_IF;
			END_IF;

		130:
			// Run macro command
			// -----------------------------------------------------------------
			m_macro.Run.Name := Parameters.MacroName;
			m_cmd.Input.MacroRun := TRUE;

			m_status.CommandDone := m_macro.Run.Done;
			m_status.CommandAcknowdledge := m_macro.Run.Acknowledge;
			m_status.CommandError := m_macro.Run.Error;
			m_status.ErrorID := m_macro.Run.ErrorID;

			IF m_var.NoCommandActive THEN
				m_sequence_state := 100;
			END_IF;

		140:
			// Save macro command
			// -----------------------------------------------------------------
			m_cmd.Input.MacroSave := TRUE;

			m_status.CommandDone := m_macro.Save.Done;
			m_status.CommandError := m_macro.Save.Error;
			m_status.ErrorID := m_macro.Save.ErrorID;

			IF m_var.NoCommandActive THEN
				m_sequence_state := 100;
			END_IF;

		150:
			// Move in plane command
			// -----------------------------------------------------------------
			m_move.MoveInPlane.Parameters := Operation.MoveInPlane;
			m_cmd.Input.MoveInPlane := TRUE;

			m_status.CommandDone := m_move.MoveInPlane.Done;
			m_status.CommandAcknowdledge := m_move.MoveInPlane.Acknowledge;
			m_status.CommandError := m_move.MoveInPlane.Error;
			m_status.ErrorID := m_move.MoveInPlane.ErrorID;

			IF m_var.NoCommandActive THEN
				m_sequence_state := 100;
			END_IF;

		160:
			// Move arc command
			// -----------------------------------------------------------------
			m_move.MoveArc.Parameters := Operation.MoveArc;
			m_cmd.Input.MoveArc := TRUE;

			m_status.CommandDone := m_move.MoveArc.Done;
			m_status.CommandAcknowdledge := m_move.MoveArc.Acknowledge;
			m_status.CommandError := m_move.MoveArc.Error;
			m_status.ErrorID := m_move.MoveArc.ErrorID;

			IF m_var.NoCommandActive THEN
				m_sequence_state := 100;
			END_IF;

		170:
			// Move short axis command
			// -----------------------------------------------------------------
			m_move.MoveShortAxis.Parameters := Operation.MoveShortAxis;
			m_cmd.Input.MoveShortAxis := TRUE;

			m_status.CommandDone := m_move.MoveShortAxis.Done;
			m_status.CommandAcknowdledge := m_move.MoveShortAxis.Acknowledge;
			m_status.CommandError := m_move.MoveShortAxis.Error;
			m_status.ErrorID := m_move.MoveShortAxis.ErrorID;

			IF m_var.NoCommandActive THEN
				m_sequence_state := 100;
			END_IF;

		180:
			// Move 6D command
			// -----------------------------------------------------------------
			m_move.Move6D.Parameters := Operation.Move6D;
			m_cmd.Input.Move6D := TRUE;

			m_status.CommandDone := m_move.Move6D.Done;
			m_status.CommandAcknowdledge := m_move.Move6D.Acknowledge;
			m_status.CommandError := m_move.Move6D.Error;
			m_status.ErrorID := m_move.Move6D.ErrorID;

			IF m_var.NoCommandActive THEN
				m_sequence_state := 100;
			END_IF;

		190:
			// Spin command
			// -----------------------------------------------------------------
			m_move.Spin.Parameters := Operation.Spin;
			m_cmd.Input.Spin := TRUE;

			m_status.CommandDone := m_move.Spin.Done;
			m_status.CommandAcknowdledge := m_move.Spin.Acknowledge;
			m_status.CommandError := m_move.Spin.Error;
			m_status.ErrorID := m_move.Spin.ErrorID;

			IF m_var.NoCommandActive THEN
				m_sequence_state := 100;
			END_IF;

		200:
			// Wait command label command
			// -----------------------------------------------------------------
			m_move.WaitCommandLabel.TriggerXID := Operation.WaitCommandLabel.TriggerShuttleID;
			m_move.WaitCommandLabel.TriggerType := Operation.WaitCommandLabel.TriggerType;
			m_move.WaitCommandLabel.TriggerCmdLb := Operation.WaitCommandLabel.TriggerCmdLb;
			m_move.WaitCommandLabel.LabelType := Operation.WaitCommandLabel.LabelType;
			m_cmd.Input.WaitCommandLabel := TRUE;

			m_status.CommandDone := m_move.WaitCommandLabel.Done;
			m_status.CommandAcknowdledge := m_move.WaitCommandLabel.Acknowledge;
			m_status.CommandError := m_move.WaitCommandLabel.Error;
			m_status.ErrorID := m_move.WaitCommandLabel.ErrorID;

			IF m_var.NoCommandActive THEN
				m_sequence_state := 100;
			END_IF;

		210:
			// Wait until all done command
			// -----------------------------------------------------------------
			FOR m_var.index := 0 TO fdSTATION_SHUTTLE_LAST_INDEX DO
				m_move.WaitUntilAllDone.Shuttles[m_var.index] := m_var.Shuttles.List[m_var.index].Shuttle6D;
			END_FOR;
			m_cmd.Input.WaitUntilAllDone := TRUE;

			m_status.CommandDone := m_move.WaitUntilAllDone.Done;
			m_status.CommandError := m_move.WaitUntilAllDone.Error;

			IF m_var.NoCommandActive THEN
				m_sequence_state := 100;
			END_IF;

		220:
			// Group couple command
			// -----------------------------------------------------------------
			m_group.CoupleCtrl.Parameters.Option := mcACP6D_SH_GROUP_COUPLE;
			m_group.CoupleCtrl.Parameters.Mode := mcACP6D_SH_GROUP_CMN_ROT_REF;
			m_cmd.Input.Group.Couple_CommonCenterPoint := TRUE;

			m_status.CommandDone := m_group.CoupleCtrl.Done;
			m_status.CommandError := m_group.CoupleCtrl.Error;
			m_status.ErrorID := m_group.CoupleCtrl.ErrorID;

			IF m_var.NoCommandActive THEN
				m_sequence_state := 100;
			END_IF;
		221:
			// Group couple command
			// -----------------------------------------------------------------
			m_group.CoupleCtrl.Parameters.Option := mcACP6D_SH_GROUP_COUPLE;
			m_group.CoupleCtrl.Parameters.Mode := mcACP6D_SH_GROUP_INDV_ROT_REF;
			m_cmd.Input.Group.Couple_OwnCenterPoint := TRUE;

			m_status.CommandDone := m_group.CoupleCtrl.Done;
			m_status.CommandError := m_group.CoupleCtrl.Error;
			m_status.ErrorID := m_group.CoupleCtrl.ErrorID;

			IF m_var.NoCommandActive THEN
				m_sequence_state := 100;
			END_IF;

		230:
			// Group decouple command
			// -----------------------------------------------------------------
			m_group.CoupleCtrl.Parameters.Option := mcACP6D_SH_GROUP_DECOUPLE;
			m_cmd.Input.Group.Decouple := TRUE;

			m_status.CommandDone := m_group.CoupleCtrl.Done;
			m_status.CommandError := m_group.CoupleCtrl.Error;
			m_status.ErrorID := m_group.CoupleCtrl.ErrorID;

			IF m_var.NoCommandActive THEN
				m_sequence_state := 100;
			END_IF;

		240:
			// Sun planet couple command
			// -----------------------------------------------------------------
			FOR m_var.index := 0 TO fdSTATION_SHUTTLE_LAST_INDEX DO
				m_move.SunPlanet.Parameters.ShuttleList[m_var.index].Shuttle := ADR(m_var.Shuttles.List[m_var.index].Shuttle6D);
			END_FOR;

			m_move.SunPlanet.Parameters.Option := mcACP6D_PLANET_ADD_SH;
			m_cmd.Input.SunPlanet.Couple := TRUE;

			m_status.CommandDone := m_move.SunPlanet.Done;
			m_status.CommandError := m_move.SunPlanet.Error;
			m_status.ErrorID := m_move.SunPlanet.ErrorID;

			IF m_var.NoCommandActive THEN
				m_sequence_state := 100;
			END_IF;

		250:
			// Sun planet decouple command
			// -----------------------------------------------------------------
			FOR m_var.index := 0 TO fdSTATION_SHUTTLE_LAST_INDEX DO
				m_move.SunPlanet.Parameters.ShuttleList[m_var.index].Shuttle := ADR(m_var.Shuttles.List[m_var.index].Shuttle6D);
			END_FOR;

			m_move.SunPlanet.Parameters.Option := mcACP6D_PLANET_REMOVE_SH;
			m_cmd.Input.SunPlanet.Decouple := TRUE;

			m_status.CommandDone := m_move.SunPlanet.Done;
			m_status.CommandError := m_move.SunPlanet.Error;
			m_status.ErrorID := m_move.SunPlanet.ErrorID;

			IF m_var.NoCommandActive THEN
				m_sequence_state := 100;
			END_IF;

END_CASE;

	// Sequence step change event
	// ----------------------------------------------------------------------------------------
	IF m_sequence_state <> m_var.SequenceStatePrevious THEN
		IF m_sequence_state = 2000 THEN
			m_var.ErroredSequenceState := m_var.SequenceStatePrevious;
		ELSE
			m_var.ErroredSequenceState := 0;
		END_IF;

		m_var.SequenceStatePrevious := m_sequence_state;
		brsmemset(ADR(m_cmd), 0, SIZEOF(m_cmd));
		brsmemset(ADR(m_status), 0, SIZEOF(m_status));
	END_IF;

	// Command label handling
	// ----------------------------------------------------------------------------------------
	IF Operation.CommandLabel.ManualMode THEN
		// Set command label from input parameters
		m_var.CommandLabel := Operation.CommandLabel.Label;
	ELSE
		// If manual mode is not on set command label automatically based on current state
		m_var.CommandLabel := State;
	END_IF;

	// Station control
	// ----------------------------------------------------------------------------------------
	m_control.StationControl.MpLink := ADR(TrafficManager);
	m_control.StationControl.Enable := Enable;
	m_control.StationControl.Station := ADR(Station);
	m_control.StationControl.To := ADR(NextStation);
	m_control.StationControl.ErrorReset := m_cmd.Input.ErrorReset;
	m_control.StationControl.Release := m_control.StationQueueControl.ReleaseShuttle;
	m_control.StationControl();

	m_control.StationQueueControl.Enable := Active;
	m_control.StationQueueControl.ShuttleList := m_var.Shuttles.List;
	m_control.StationQueueControl.ShuttleCapacity := Parameters.ShuttleCapacity;
	m_control.StationQueueControl.ReleaseShuttles := m_cmd.Input.ReleaseAllShuttles;
	m_control.StationQueueControl.pStation := ADR(m_control.StationControl);
	m_control.StationQueueControl();

	m_control.VirtualShuttleCreate.Execute := m_cmd.VirtualShuttleCreate;
	m_control.VirtualShuttleCreate.Assembly := ADR(Assembly);
	m_control.VirtualShuttleCreate();

	m_control.GetShuttleInfo.Execute := m_cmd.GetShuttleInfo;
	m_control.GetShuttleInfo();

	// Movement
	// ----------------------------------------------------------------------------------------
	m_move.MoveInPlane.Execute := m_cmd.Input.MoveInPlane;
	m_move.MoveInPlane.Shuttle := ADR(Operation.Shuttle.Shuttle6D);
	m_move.MoveInPlane.CommandLabel := m_var.CommandLabel;
	m_move.MoveInPlane();

	m_move.MoveArc.Execute := m_cmd.Input.MoveArc;
	m_move.MoveArc.Shuttle := ADR(Operation.Shuttle.Shuttle6D);
	m_move.MoveArc.CommandLabel := m_var.CommandLabel;
	m_move.MoveArc();

	m_move.Move6D.Execute := m_cmd.Input.Move6D;
	m_move.Move6D.Shuttle := ADR(Operation.Shuttle.Shuttle6D);
	m_move.Move6D.CommandLabel := m_var.CommandLabel;
	m_move.Move6D();

	m_move.MoveShortAxis.Execute := m_cmd.Input.MoveShortAxis;
	m_move.MoveShortAxis.Shuttle := ADR(Operation.Shuttle.Shuttle6D);
	m_move.MoveShortAxis.CommandLabel := m_var.CommandLabel;
	m_move.MoveShortAxis();

	m_move.Spin.Execute := m_cmd.Input.Spin;
	m_move.Spin.Shuttle := ADR(Operation.Shuttle.Shuttle6D);
	m_move.Spin.CommandLabel := m_var.CommandLabel;
	m_move.Spin();

	m_move.WaitCommandLabel.Execute := m_cmd.Input.WaitCommandLabel;
	m_move.WaitCommandLabel.Shuttle := ADR(Operation.Shuttle.Shuttle6D);
	m_move.WaitCommandLabel.CommandLabel := m_var.CommandLabel;
	m_move.WaitCommandLabel();

	m_move.WaitUntilAllDone.Execute := m_cmd.Input.WaitUntilAllDone;
	m_move.WaitUntilAllDone();

	// Sun Planet
	// ----------------------------------------------------------------------------------------
	m_move.SunPlanet.Execute := m_cmd.Input.SunPlanet.Couple OR m_cmd.Input.SunPlanet.Decouple;
	m_move.SunPlanet.Shuttle := ADR(Operation.Shuttle.Shuttle6D);
	m_move.SunPlanet();

	// Macro
	// ----------------------------------------------------------------------------------------
	m_macro.Create.Execute := m_cmd.MacroCreate;
	m_macro.Create.Assembly := ADR(Assembly);
	m_macro.Create();

	m_macro.Delete.Execute := m_cmd.MacroDelete;
	m_macro.Delete.Assembly := ADR(Assembly);
	m_macro.Delete();

	m_macro.Save.Execute := m_cmd.Input.MacroSave;
	m_macro.Save.Shuttle := ADR(m_var.MacroShuttle.Shuttle6D);
	m_macro.Save();

	m_macro.Run.Execute := m_cmd.Input.MacroRun;
	m_macro.Run.Shuttle := ADR(Operation.Shuttle.Shuttle6D);
	m_macro.Run.CommandLabel := m_var.CommandLabel;
	m_macro.Run();

	// Zone
	// ----------------------------------------------------------------------------------------
	m_zone.Create.Execute := m_cmd.ZoneCreate;
	m_zone.Create.Assembly := ADR(Assembly);
	m_zone.Create();

	m_zone.Find.Execute := m_cmd.ZoneFind;
	m_zone.Find.Assembly := ADR(Assembly);
	m_zone.Find();

	m_zone.GetBarrierInfo.Execute := m_cmd.ZoneGetBarrierInfo;
	m_zone.GetBarrierInfo.Zone := ADR(m_zone.Zone);
	m_zone.GetBarrierInfo();

	// Group
	// ----------------------------------------------------------------------------------------
	m_group.Create.Execute := m_cmd.GroupCreate;
	m_group.Create.Assembly := ADR(Assembly);
	m_group.Create();

	m_group.Clear.Execute := m_cmd.GroupClear;
	m_group.Clear.ShuttleGroup := ADR(m_var.ShuttleGroup);
	m_group.Clear();

	m_group.AddShuttle.Execute := m_cmd.GroupAddShuttle;
	m_group.AddShuttle.ShuttleGroup := ADR(m_var.ShuttleGroup);
	m_group.AddShuttle();

	m_group.CoupleCtrl.Execute := m_cmd.Input.Group.Couple_CommonCenterPoint OR m_cmd.Input.Group.Couple_OwnCenterPoint OR m_cmd.Input.Group.Decouple;
	m_group.CoupleCtrl.ShuttleGroup := ADR(m_var.ShuttleGroup);
	m_group.CoupleCtrl();

	m_group.Delete.Execute := m_cmd.GroupDelete;
	m_group.Delete.ShuttleGroup := ADR(m_var.ShuttleGroup);
	m_group.Delete();

	// Station outputs
	// ----------------------------------------------------------------------------------------
	Shuttles := m_var.Shuttles;
	MacroShuttle := m_var.MacroShuttle;
	NumOccupyingShuttles := m_control.StationControl.Info.NumOccupyingShuttles;

	CommandDone := m_status.CommandDone;
	CommandAcknowledge := m_status.CommandAcknowdledge;
	CommandError := m_status.CommandError;
	ErrorID := m_status.ErrorID;
	ErroredSequenceState := m_var.ErroredSequenceState;

END_FUNCTION_BLOCK
```

### global.var
```iecst
VAR
	gFastDemo : FastDemoType := (0);
END_VAR
```

### global.typ
```iecst
(*
Program: FastDemo

Description
(short summary)

*)
(*========== INPUTS ==========*)

TYPE
	FastDemoInputCommandType : 	STRUCT
		Activate : BOOL;
	END_STRUCT;
	FastDemoInputStatusType : 	STRUCT
		SetupComplete : BOOL;
	END_STRUCT;
	FastDemoInputType : 	STRUCT
		Force : BOOL;
		Command : FastDemoInputCommandType;
		Status : FastDemoInputStatusType;
	END_STRUCT;
END_TYPE

(*========== OUTPUTS ==========*)

TYPE
	FastDemoOutputCommandType : 	STRUCT
		NewCommand : BOOL;
	END_STRUCT;
	FastDemoOutputStatusType : 	STRUCT
		NewStatus : BOOL;
	END_STRUCT;
	FastDemoOutputType : 	STRUCT
		Command : FastDemoOutputCommandType;
		Status : FastDemoOutputStatusType;
	END_STRUCT;
END_TYPE

(*========== ERRORS ==========*)
(*========== SETTINGS ==========*)

TYPE
	FastDemoSettingsType : 	STRUCT
		Enable : BOOL;
	END_STRUCT;
END_TYPE

(*========== INTERFACE ==========*)

TYPE
	FastDemoType : 	STRUCT
		Error : GeneralErrorInfoType;
		Input : FastDemoInputType;
		Output : FastDemoOutputType;
		Settings : FastDemoSettingsType;
	END_STRUCT;
END_TYPE
```

### Program Logical/src/FastDemo/FastDemo (IEC)

#### FastDemo.st
```iecst
PROGRAM _INIT

    // Access the task interface
    task ACCESS ADR(gFastDemo);

    // Register module config interface for common setup/parametrization functionality
    //fb.MpRecipeRegPar_settings(MpLink := ADR(gSystemSettings), Enable := TRUE , PVName := ADR('gFastDemo.settings'), Category := ADR('FastDemo'));

    // Check for simulator
    //task.IsSimulated := DiagCpuIsSimulated();

    // PackML setup
    // =================================================================================================================
    em.Setup.Name := 'FastDemo';
	em.Setup.ParentName := 'Main';

END_PROGRAM

PROGRAM _CYCLIC

    // Access task interface
    // =================================================================================================================
    task ACCESS ADR(gFastDemo);

    // Inputs
    // =================================================================================================================
    IF NOT task.Input.Force THEN

	END_IF

	// Issue 1: Multiple recovery points do not work correctly
	// =================================================================================================================
	CASE issue1.state OF
		1:
			fb.TrafficControl.Recover := TRUE;
			IF fb.TrafficControl.RecoverDone THEN
				fb.TrafficControl.Recover := FALSE;
				issue1.state := 2;
			END_IF;
		2:
			fb.TrafficControl.ActivateRecipe := TRUE;
			IF fb.TrafficControl.ActivateRecipeDone THEN
				fb.TrafficControl.ActivateRecipe := FALSE;
				issue1.state := 3;
			END_IF;
		ELSE
			fb.TrafficControl.Recover := FALSE;
			fb.TrafficControl.ActivateRecipe := FALSE;
	END_CASE;

	// Issue 2: Wait for command label command does not work correctly
	// =================================================================================================================

	// Issue 3: Move Async error after group rotate stop
	// =================================================================================================================

	// Task state machine
	// =================================================================================================================
	// PackML state machine execution
	PackML_state_machine;

	// Detect state change events
	// =================================================================================================================
	// Record information which state caused abort
	fb.R_TRIG_Abort(CLK := em.Command.Abort);

	IF fb.R_TRIG_Abort.Q THEN
		task.Error.State := em.StateCurrent;
		task.Error.SubState := em.SubState;
		task.Error.Description := em.StateInfo;
	END_IF;

	// State change event
	fb.rtStateComplete(CLK := em.Command.StateComplete);

	IF fb.rtStateComplete.Q THEN
		em.StateInfo := '';
		brsmemset(ADR(actions_state), 0, SIZEOF(actions_state));

		// Record information which state caused abort
		IF em.StateCurrent = STATE_ABORTING THEN
			task.Error.State := local.lastState;
			task.Error.SubState := local.lastSubState;
			task.Error.Description := local.lastStateInfo;
		END_IF;
	END_IF;

	// Substate changed event
	IF em.SubState <> local.lastSubState THEN
		em.StateInfo := '';
		brsmemset(ADR(actions_substate), 0, SIZEOF(actions_substate));
		local.lastSubState := em.SubState;
	END_IF;

	// PackML equipment module
	// =================================================================================================================
	em();

	// Function calls
    // =================================================================================================================
	fb.TrafficControl.Enable := TRUE;
	fb.TrafficControl.MpLink := ADR(TrafficManager_x6d_1);
//	fb.TrafficControl.ActivateRecipe := actions_substate.traffic_activate_recipe;
//	fb.TrafficControl.DeactivateRecipe := actions_substate.traffic_deactivate_recipe;
//	fb.TrafficControl.ErrorReset := actions_state.error_reset;
//	fb.TrafficControl.Halt := actions_substate.traffic_halt;
//	fb.TrafficControl.Recover := actions_substate.traffic_recover;
//	fb.TrafficControl.Resume := actions_substate.traffic_resume;
//	fb.TrafficControl.Stop := actions_substate.traffic_stop;
	fb.TrafficControl();

	fb.TON_RecoverTimeout.IN := fb.TrafficControl.RecoverBuffered;
	fb.TON_RecoverTimeout.PT := T#5s;
	fb.TON_RecoverTimeout();

	fb.TrafficMonitor.Enable := TRUE;
	fb.TrafficMonitor.MpLink := ADR(TrafficManager_x6d_1);
	fb.TrafficMonitor();

	// Station logic calls
	FOR station_num := 0 TO STATION_COUNT DO
		station ACCESS ADR(stations[station_num]);

		station.Enable := actions_state.activate_stations;
		station.Parameters.StationNumber := station_num;
		station.Assembly := ADR(gAssembly6D_Big);
		station.TrafficManager := ADR(TrafficManager_x6d_1);
		station();
	END_FOR

	// Task outputs
	// =================================================================================================================

	// Task diagnostics
	// =================================================================================================================
	gTasks.FastDemo.State := em.StateCurrent;
	gTasks.FastDemo.SubState := em.SubState;
	gTasks.FastDemo.Mode := em.ModeID;
	gTasks.FastDemo.StateComplete := em.Command.StateComplete;
	gTasks.FastDemo.StateInfo := em.StateInfo;
	gTasks.FastDemo.WaitingForTask := em.Info.WaitingFor.Name;
	gTasks.FastDemo.Error := task.Error;

END_PROGRAM

PROGRAM _EXIT

END_PROGRAM
```

#### local.typ
```iecst
TYPE
	FastDemoFbType : 	STRUCT
		MpRecipeRegPar_settings : BOOL;
		TrafficControl : MpTrafficControl;
		TrafficMonitor : MpTrafficMonitor;
		rtStateComplete : R_TRIG;
		R_TRIG_Abort : R_TRIG;
		TON_RecoverTimeout : TON;
	END_STRUCT;
	FastDemoLocalType : 	STRUCT
		lastState : DINT;
		lastSubState : DINT;
		lastStateInfo : STRING[80];
		allStationsDeactivated : BOOL;
	END_STRUCT;
	FastDemoActionsStateType : 	STRUCT
		error_reset : BOOL;
		activate_stations : BOOL;
	END_STRUCT;
	FastDemoActionsSubstateType : 	STRUCT
		traffic_activate_recipe : BOOL; (*Task actions are not automatically reset*)
		traffic_deactivate_recipe : BOOL; (*Task actions are not automatically reset*)
		traffic_halt : BOOL;
		traffic_recover : BOOL;
		traffic_resume : BOOL;
		traffic_stop : BOOL;
	END_STRUCT;
	FastDemoHmiType : 	STRUCT
		isRunning : BOOL;
	END_STRUCT;
END_TYPE

(*Insert your comment here.*)

TYPE
	Issue1Type : 	STRUCT
		state : USINT;
	END_STRUCT;
END_TYPE
```

#### local.var
```iecst
VAR
	task : REFERENCE TO FastDemoType;
	local : FastDemoLocalType;
	fb : FastDemoFbType;
	hmi : FastDemoHmiType;
	actions_state : FastDemoActionsStateType;
	actions_substate : FastDemoActionsSubstateType;
END_VAR
(* ----- PackML ----- *)
VAR
	em : EquipmentModule;
END_VAR
(*----- Stations ----*)
VAR
	station_num : {REDUND_UNREPLICABLE} DINT := 0;
	str : STRING[80];
	i : DINT;
END_VAR
VAR CONSTANT
	STATION_COUNT : DINT := 7;
END_VAR
VAR
	stations : ARRAY[0..STATION_COUNT] OF fdStation;
	station : REFERENCE TO fdStation;
END_VAR
(*Issue 1*)
VAR
	issue1 : Issue1Type;
END_VAR
```

#### PackML.st
```iecst
// PackML state machine. Split into different sections that handle
// different logical sequences of PackML stadards' steps
// INFO: Add mode specific code into states by adding CASE structure
// 	CASE em.ModeID OF
//		MODE_PRODUCTION:
//			*CODE*;
//		MODE_MAINTENANCE:
//			*CODE*;
//		MODE_MANUAL:
//			*CODE*;
//		END_CASE
// -----------------------------------------------------------------

ACTION PackML_state_machine:
	// =================================================================================================================
    // Global PackML events
    // =================================================================================================================

    // =================================================================================================================
    // Normal work sequence
    // =================================================================================================================
    CASE em.StateCurrent OF
        STATE_STOPPED:
            em.StateInfo := '';
            // -----------------------------------------------------------------
            em.Command.StateComplete := TRUE;

        STATE_RESETTING:
			CASE em.SubState OF
				0:
					em.StateInfo := 'Reset traffic control errors';
					// -----------------------------------------------------------------
					actions_state.error_reset := TRUE;
					IF NOT fb.TrafficControl.Error THEN
	  					em.SubState := 10;
					END_IF;
				10:
					em.StateInfo := 'Wait until all stations are deactivated';
					// -----------------------------------------------------------------
					local.allStationsDeactivated := TRUE;

					FOR station_num := 0 TO STATION_COUNT DO
						station ACCESS ADR(stations[station_num]);

						IF station.Active THEN
							local.allStationsDeactivated := FALSE;
							EXIT;
						END_IF;
					END_FOR;

					IF local.allStationsDeactivated THEN
	  					em.SubState := 100;
					END_IF;

				100:
					em.StateInfo := 'Reset complete';
					// -----------------------------------------------------------------
					em.Command.StateComplete := TRUE;
			END_CASE;

		STATE_IDLE:
			em.StateInfo := '';
			// -----------------------------------------------------------------
			em.Command.StateComplete := TRUE;

		STATE_STARTING:
			CASE em.SubState OF
				0:
					em.StateInfo := 'Move shuttles to recovery points';
					// -----------------------------------------------------------------
					fb.TrafficControl.Velocity := 1.8;
					fb.TrafficControl.Acceleration := 8.0;
					actions_substate.traffic_recover := TRUE;

					IF fb.TrafficControl.RecoverDone OR fb.TON_RecoverTimeout.Q THEN
						em.SubState := 10;
					END_IF;
				10:
					em.StateInfo := 'Activating traffic recipe';
					// -----------------------------------------------------------------
					actions_substate.traffic_activate_recipe := TRUE;

					IF fb.TrafficControl.ActivateRecipeDone THEN
						em.SubState := 100;
					END_IF;
				100:
					em.StateInfo := 'Traffic manager started';
					// -----------------------------------------------------------------
					IF fb.TrafficControl.Error THEN
	  					em.SubState := 200;
					ELSE
						em.Command.StateComplete := TRUE;
					END_IF;
			END_CASE;

        STATE_EXECUTE:
            em.StateInfo := 'Running feature demo';
            // -----------------------------------------------------------------
			em.Command.StateComplete := TRUE;

			actions_state.activate_stations := TRUE;

//			execute_station_S1;
//			execute_station_S2;
//			execute_station_S3;
//			execute_station_S4;
//			execute_station_S5;
//			execute_station_S6;
			//execute_station_S7;

        STATE_COMPLETING:
            em.StateInfo := '';
            // -----------------------------------------------------------------
            em.Command.StateComplete := TRUE;

        STATE_COMPLETED:
            em.StateInfo := '';
            // -----------------------------------------------------------------
            em.Command.StateComplete := TRUE;

        STATE_STOPPING:
            em.StateInfo := 'Stop traffic manager';
			// -----------------------------------------------------------------
			actions_substate.traffic_stop := TRUE;
			IF fb.TrafficControl.StopDone THEN
	  			em.Command.StateComplete := TRUE;
			END_IF;
	END_CASE

    // =================================================================================================================
    // Module activation sequence
    // =================================================================================================================
    CASE em.StateCurrent OF
        STATE_DEACTIVATING:
            em.StateInfo := '';
            // -----------------------------------------------------------------
            em.Command.StateComplete := TRUE;

        STATE_DEACTIVATED:
            em.StateInfo := '';
            // -----------------------------------------------------------------
            em.Command.StateComplete := TRUE;

        STATE_ACTIVATING:
            em.StateInfo := '';
            // -----------------------------------------------------------------
            em.Command.StateComplete := TRUE;

    END_CASE

    // =================================================================================================================
    // Abort sequence
    // =================================================================================================================
    CASE em.StateCurrent OF
        STATE_ABORTING:
            em.StateInfo := '';
            // -----------------------------------------------------------------
            em.Command.StateComplete := TRUE;

        STATE_ABORTED:
            em.StateInfo := '';
            // -----------------------------------------------------------------
            em.Command.StateComplete := TRUE;

        STATE_CLEARING:
            em.StateInfo := '';
            // -----------------------------------------------------------------
            em.Command.StateComplete := TRUE;
    END_CASE

    // =================================================================================================================
    // Hold sequence
    // =================================================================================================================
    CASE em.StateCurrent OF
        STATE_HOLDING:
            em.StateInfo := '';
            // -----------------------------------------------------------------
            em.Command.StateComplete := TRUE;

        STATE_HELD:
            em.StateInfo := '';
            // -----------------------------------------------------------------
            em.Command.StateComplete := TRUE;

        STATE_UNHOLDING:
            em.StateInfo := '';
            // -----------------------------------------------------------------
            em.Command.StateComplete := TRUE;
    END_CASE

    // =================================================================================================================
    // Suspend sequence
    // =================================================================================================================
    CASE em.StateCurrent OF
        STATE_SUSPENDING:
            em.StateInfo := '';
            // -----------------------------------------------------------------
            em.Command.StateComplete := TRUE;

        STATE_SUSPENDED:
            em.StateInfo := '';
            // -----------------------------------------------------------------
            em.Command.StateComplete := TRUE;

        STATE_UNSUSPENDING:
            em.StateInfo := '';
            // -----------------------------------------------------------------
            em.Command.StateComplete := TRUE;

    END_CASE

END_ACTION
```

#### defaults.st
```iecst
ACTION set_movement_parameters_to_default_values:
	// Move in plane
	brsmemset(ADR(station.Operation.MoveInPlane), 0, SIZEOF(station.Operation.MoveInPlane));
	station.Operation.MoveInPlane.Velocity := 1.5;
	station.Operation.MoveInPlane.Acceleration := 18;
	station.Operation.MoveInPlane.EndVelocity := 0;
	station.Operation.MoveInPlane.Path := mcACP6D_PATH_DIRECT;
	station.Operation.MoveInPlane.Mode := mcACP6D_MOVE_ABSOLUTE;

	// Move short axis
	brsmemset(ADR(station.Operation.MoveShortAxis), 0, SIZEOF(station.Operation.MoveShortAxis));
	station.Operation.MoveShortAxis.Velocity.Rx := 0.1;
	station.Operation.MoveShortAxis.Velocity.Ry := 0.1;
	station.Operation.MoveShortAxis.Velocity.Rz := 0.1;
	station.Operation.MoveShortAxis.Velocity.Z := 0.005;
	station.Operation.MoveShortAxis.Position.Rx := 0;
	station.Operation.MoveShortAxis.Position.Ry:= 0;
	station.Operation.MoveShortAxis.Position.Rz := 0;
	station.Operation.MoveShortAxis.Position.Z := gDEFAULT_Z;
	station.Operation.MoveShortAxis.Mode := mcACP6D_MOVE_ABSOLUTE;

	// Move arc
	brsmemset(ADR(station.Operation.MoveArc), 0, SIZEOF(station.Operation.MoveArc));
	station.Operation.MoveArc.Velocity := 1.5;
	station.Operation.MoveArc.Acceleration := 18;
	station.Operation.MoveArc.EndVelocity := 0;
	station.Operation.MoveArc.Angular.Angle := 0;
	station.Operation.MoveArc.Option := mcACP6D_ARC_ANGULAR;
	station.Operation.MoveArc.Mode :=  mcACP6D_MOVE_RELATIVE;

	// Move 6D
	brsmemset(ADR(station.Operation.Move6D), 0, SIZEOF(station.Operation.Move6D));

	// Wait command label
	station.Operation.WaitCommandLabel.LabelType :=  mcACP6D_SH_WAIT_CMDLB_REGULAR;
	station.Operation.WaitCommandLabel.TriggerCmdLb := 0;
	station.Operation.WaitCommandLabel.TriggerType := mcACP6D_SH_WAIT_CMDLB_START;
	station.Operation.WaitCommandLabel.TriggerShuttleID := 0;

END_ACTION
```

#### station_S1.st
```iecst
ACTION execute_station_S1:
	// Point station reference to this station
	station ACCESS ADR(stations[1]);

	// Station parameters
	station.Station := ADR(S1);
	station.NextStation := ADR(S2);
	station.Parameters.ShuttleCapacity := 1;
	station.Parameters.Zone.BottomLeft.X := 0;
	station.Parameters.Zone.BottomLeft.Y := 0;
	station.Parameters.Zone.TopRight.X := 0.240;
	station.Parameters.Zone.TopRight.Y := 0.480;

	CASE station.State OF
		0:
			station.StateInfo := 'Activating station';
			// -----------------------------------------------------------------
			IF station.Active THEN
				station.Loop := 0;
				station.JumpToState := 100;
			END_IF;

		100:
			station.StateInfo := 'Movement settings';
			// -----------------------------------------------------------------
			set_movement_parameters_to_default_values;
			station.Operation.Shuttle := station.MacroShuttle;
			station.NextState := TRUE;
		101:
			station.StateInfo := 'Move to UL';
			// -----------------------------------------------------------------
			station.Operation.MoveInPlane.Position.X := 0.060;
			station.Operation.MoveInPlane.Position.Y := 0.420;
			station.Commands.MoveInPlane := TRUE;

			IF station.CommandAcknowledge THEN
				station.NextState := TRUE;
			END_IF;
		102:
			station.StateInfo := 'Move to LL';
			// -----------------------------------------------------------------
			station.Operation.MoveInPlane.Mode := mcACP6D_MOVE_ABSOLUTE;
			station.Operation.MoveInPlane.Position.X := 0.060;
			station.Operation.MoveInPlane.Position.Y := 0.060;
			station.Commands.MoveInPlane := TRUE;

			IF station.CommandAcknowledge THEN
				station.NextState := TRUE;
			END_IF;
		103:
			station.StateInfo := 'Move to LR';
			// -----------------------------------------------------------------
			station.Operation.MoveInPlane.Mode := mcACP6D_MOVE_ABSOLUTE;
			station.Operation.MoveInPlane.Position.X := 0.180;
			station.Operation.MoveInPlane.Position.Y := 0.060;
			station.Commands.MoveInPlane := TRUE;

			IF station.CommandAcknowledge THEN
				station.NextState := TRUE;
			END_IF;
		104:
			station.StateInfo := 'Move to UR';
			// -----------------------------------------------------------------
			station.Operation.MoveInPlane.Mode := mcACP6D_MOVE_ABSOLUTE;
			station.Operation.MoveInPlane.Position.X := 0.180;
			station.Operation.MoveInPlane.Position.Y := 0.420;
			station.Commands.MoveInPlane := TRUE;

			IF station.CommandAcknowledge THEN
				station.NextState := TRUE;
			END_IF;
		105:
			station.StateInfo := 'Move to UL';
			// -----------------------------------------------------------------
			station.Operation.MoveInPlane.Mode := mcACP6D_MOVE_ABSOLUTE;
			station.Operation.MoveInPlane.Position.X := 0.060;
			station.Operation.MoveInPlane.Position.Y := 0.420;
			station.Commands.MoveInPlane := TRUE;

			IF station.CommandAcknowledge THEN
				station.NextState := TRUE;
			END_IF;
		106:
			station.StateInfo := 'Move to LR';
			// -----------------------------------------------------------------
			station.Operation.MoveInPlane.Mode := mcACP6D_MOVE_ABSOLUTE;
			station.Operation.MoveInPlane.Position.X := 0.180;
			station.Operation.MoveInPlane.Position.Y := 0.060;
			station.Commands.MoveInPlane := TRUE;

			IF station.CommandAcknowledge THEN
				station.NextState := TRUE;
			END_IF;
		107:
			station.StateInfo := 'Move to LL';
			// -----------------------------------------------------------------
			station.Operation.MoveInPlane.Mode := mcACP6D_MOVE_ABSOLUTE;
			station.Operation.MoveInPlane.Position.X := 0.060;
			station.Operation.MoveInPlane.Position.Y := 0.060;
			station.Commands.MoveInPlane := TRUE;

			IF station.CommandAcknowledge THEN
				station.NextState := TRUE;
			END_IF;
		108:
			station.StateInfo := 'Move to UR';
			// -----------------------------------------------------------------
			station.Operation.MoveInPlane.Mode := mcACP6D_MOVE_ABSOLUTE;
			station.Operation.MoveInPlane.Position.X := 0.180;
			station.Operation.MoveInPlane.Position.Y := 0.420;
			station.Commands.MoveInPlane := TRUE;

			IF station.CommandAcknowledge THEN
				station.NextState := TRUE;
			END_IF;
		109:
			station.StateInfo := 'Move to UL';
			// -----------------------------------------------------------------
			station.Operation.MoveInPlane.Mode := mcACP6D_MOVE_ABSOLUTE;
			station.Operation.MoveInPlane.Position.X := 0.060;
			station.Operation.MoveInPlane.Position.Y := 0.420;
			station.Commands.MoveInPlane := TRUE;

			IF station.CommandAcknowledge THEN
				station.NextState := TRUE;
			END_IF;
		110:
			station.StateInfo := 'Move to LL';
			// -----------------------------------------------------------------
			station.Operation.MoveInPlane.Mode := mcACP6D_MOVE_ABSOLUTE;
			station.Operation.MoveInPlane.Position.X := 0.060;
			station.Operation.MoveInPlane.Position.Y := 0.060;
			station.Commands.MoveInPlane := TRUE;

			IF station.CommandAcknowledge THEN
				station.NextState := TRUE;
			END_IF;
		111:
			station.StateInfo := 'Move right';
			// -----------------------------------------------------------------
			station.Operation.MoveInPlane.Mode := mcACP6D_MOVE_RELATIVE;
			station.Operation.MoveInPlane.Position.X := 0.120;
			station.Operation.MoveInPlane.Position.Y := 0.000;
			station.Commands.MoveInPlane := TRUE;

			IF station.CommandAcknowledge THEN
				station.NextState := TRUE;
			END_IF;
		112:
			station.StateInfo := 'Move up';
			// -----------------------------------------------------------------
			station.Operation.MoveInPlane.Mode := mcACP6D_MOVE_RELATIVE;
			station.Operation.MoveInPlane.Position.X := 0.000;
			station.Operation.MoveInPlane.Position.Y := 0.120;
			station.Commands.MoveInPlane := TRUE;

			IF station.CommandAcknowledge THEN
				station.NextState := TRUE;
			END_IF;
		113:
			station.StateInfo := 'Move left';
			// -----------------------------------------------------------------
			station.Operation.MoveInPlane.Mode := mcACP6D_MOVE_RELATIVE;
			station.Operation.MoveInPlane.Position.X := - 0.120;
			station.Operation.MoveInPlane.Position.Y := 0.000;
			station.Commands.MoveInPlane := TRUE;

			IF station.CommandAcknowledge THEN
				station.NextState := TRUE;
			END_IF;
		114:
			station.StateInfo := 'Move up';
			// -----------------------------------------------------------------
			station.Operation.MoveInPlane.Mode := mcACP6D_MOVE_RELATIVE;
			station.Operation.MoveInPlane.Position.X := 0.000;
			station.Operation.MoveInPlane.Position.Y := 0.120;
			station.Commands.MoveInPlane := TRUE;

			IF station.CommandAcknowledge THEN
				station.NextState := TRUE;
			END_IF;
		115:
			station.StateInfo := 'Move right';
			// -----------------------------------------------------------------
			station.Operation.MoveInPlane.Mode := mcACP6D_MOVE_RELATIVE;
			station.Operation.MoveInPlane.Position.X := 0.120;
			station.Operation.MoveInPlane.Position.Y := 0.000;
			station.Commands.MoveInPlane := TRUE;

			IF station.CommandAcknowledge THEN
				station.NextState := TRUE;
			END_IF;
		116:
			station.StateInfo := 'Move up';
			// -----------------------------------------------------------------
			station.Operation.MoveInPlane.Mode := mcACP6D_MOVE_RELATIVE;
			station.Operation.MoveInPlane.Position.X := 0.000;
			station.Operation.MoveInPlane.Position.Y := 0.120;
			station.Commands.MoveInPlane := TRUE;

			IF station.CommandAcknowledge THEN
				station.NextState := TRUE;
			END_IF;
		117:
			station.StateInfo := 'Move left';
			// -----------------------------------------------------------------
			station.Operation.MoveInPlane.Mode := mcACP6D_MOVE_RELATIVE;
			station.Operation.MoveInPlane.Position.X := - 0.120;
			station.Operation.MoveInPlane.Position.Y := 0.000;
			station.Commands.MoveInPlane := TRUE;

			IF station.CommandAcknowledge THEN
				station.NextState := TRUE;
			END_IF;
		118:
			station.StateInfo := 'Move down';
			// -----------------------------------------------------------------
			station.Operation.MoveInPlane.Mode := mcACP6D_MOVE_RELATIVE;
			station.Operation.MoveInPlane.Position.X := 0.000;
			station.Operation.MoveInPlane.Position.Y := - 0.120;
			station.Commands.MoveInPlane := TRUE;

			IF station.CommandAcknowledge THEN
				station.NextState := TRUE;
			END_IF;
		119:
			station.StateInfo := 'Move right';
			// -----------------------------------------------------------------
			station.Operation.MoveInPlane.Mode := mcACP6D_MOVE_RELATIVE;
			station.Operation.MoveInPlane.Position.X := 0.120;
			station.Operation.MoveInPlane.Position.Y := 0.000;
			station.Commands.MoveInPlane := TRUE;

			IF station.CommandAcknowledge THEN
				station.NextState := TRUE;
			END_IF;
		120:
			station.StateInfo := 'Move down';
			// -----------------------------------------------------------------
			station.Operation.MoveInPlane.Mode := mcACP6D_MOVE_RELATIVE;
			station.Operation.MoveInPlane.Position.X := 0.000;
			station.Operation.MoveInPlane.Position.Y := - 0.120;
			station.Commands.MoveInPlane := TRUE;

			IF station.CommandAcknowledge THEN
				station.NextState := TRUE;
			END_IF;
		121:
			station.StateInfo := 'Move left';
			// -----------------------------------------------------------------
			station.Operation.MoveInPlane.Mode := mcACP6D_MOVE_RELATIVE;
			station.Operation.MoveInPlane.Position.X := - 0.120;
			station.Operation.MoveInPlane.Position.Y := 0.000;
			station.Commands.MoveInPlane := TRUE;

			IF station.CommandAcknowledge THEN
				station.NextState := TRUE;
			END_IF;
		122:
			station.StateInfo := 'Move down';
			// -----------------------------------------------------------------
			station.Operation.MoveInPlane.Mode := mcACP6D_MOVE_RELATIVE;
			station.Operation.MoveInPlane.Position.X := 0.000;
			station.Operation.MoveInPlane.Position.Y := - 0.120;
			station.Commands.MoveInPlane := TRUE;

			IF station.CommandAcknowledge THEN
				station.NextState := TRUE;
			END_IF;
		123:
			station.StateInfo := 'Move right';
			// -----------------------------------------------------------------
			station.Operation.MoveInPlane.Mode := mcACP6D_MOVE_RELATIVE;
			station.Operation.MoveInPlane.Position.X := 0.120;
			station.Operation.MoveInPlane.Position.Y := 0.000;
			station.Commands.MoveInPlane := TRUE;

			IF station.CommandAcknowledge THEN
				station.JumpToState := 199;
			END_IF;
		199:
			station.StateInfo := 'Save macro';
			// -----------------------------------------------------------------
			station.Commands.MacroSave := TRUE;

			IF station.CommandDone THEN
				station.JumpToState := 200;
			END_IF;

		200:
			station.StateInfo := 'Waiting for shuttle to arrive at station';
			// -----------------------------------------------------------------
			station.Loop := 0;

			IF station.NumOccupyingShuttles > 0 THEN
				station.NextState := TRUE;
			END_IF;
		201:
			station.StateInfo := 'Add last arrived shuttle to the station';
			// -----------------------------------------------------------------
			station.Commands.AddShuttle := TRUE;

			IF station.CommandDone THEN
	 			station.NextState := TRUE;
			END_IF;
		202:
			station.StateInfo := 'Run macro';
			// -----------------------------------------------------------------
			station.Operation.Shuttle := station.Shuttles.List[0];
			station.Commands.MacroRun := TRUE;

			IF station.CommandDone THEN
				station.Loop := station.Loop + 1;
				IF station.Loop < 3 THEN
					station.Commands.MacroRun := FALSE;
				ELSE
					station.JumpToState := 1000;
				END_IF;
			END_IF;

		1000:
			station.StateInfo := 'Release shuttle to traffic network';
			// -----------------------------------------------------------------
			station.Commands.ReleaseAllShuttles := TRUE;

			IF station.CommandDone THEN
				station.JumpToState := 200;
			END_IF;
	END_CASE;

	// Add macro info for these steps
	IF station.State > 100 AND station.State < 200 THEN
		station.StateInfo := CONCAT('Writing macro - ', station.StateInfo);
	END_IF;

END_ACTION
```

#### station_S2.st
```iecst
ACTION execute_station_S2:
	// Point station reference to this station
	station ACCESS ADR(stations[2]);

	// Station parameters
	station.Station := ADR(S2);
	station.NextStation := ADR(B1);
	station.Parameters.ShuttleCapacity := 1;
	station.Parameters.Zone.BottomLeft.X := 0.720;
	station.Parameters.Zone.BottomLeft.Y := 0;
	station.Parameters.Zone.TopRight.X := 0.960;
	station.Parameters.Zone.TopRight.Y := 0.480;

	CASE station.State OF
		0:
			station.StateInfo := 'Activating station';
			// -----------------------------------------------------------------
			IF station.Active THEN
				station.Loop := 0;
				station.JumpToState := 100;
			END_IF;

		100:
			station.StateInfo := 'Movement settings';
			// -----------------------------------------------------------------
			set_movement_parameters_to_default_values;

			station.Operation.Shuttle := station.MacroShuttle;
			station.Operation.Spin.Acceleration := 35.0;
			station.Operation.Spin.Angle := 0;
			station.Operation.Spin.Duration := 2.0;

			station.NextState := TRUE;
		101:
			station.StateInfo := 'Move to position 1';
			// -----------------------------------------------------------------
			station.Operation.MoveInPlane.Mode := mcACP6D_MOVE_ABSOLUTE;
			station.Operation.MoveInPlane.Position.X := 0.840;
			station.Operation.MoveInPlane.Position.Y := 0.120;

			station.Commands.MoveInPlane := TRUE;

			IF station.CommandAcknowledge THEN
				station.NextState := TRUE;
			END_IF;
		102:
			station.StateInfo := 'Spin 1';
			// -----------------------------------------------------------------
			station.Operation.Spin.Velocity := 22.0;
			station.Commands.Spin := TRUE;

			IF station.CommandAcknowledge THEN
				station.NextState := TRUE;
			END_IF;
		103:
			station.StateInfo := 'Move position 2';
			// -----------------------------------------------------------------
			station.Operation.MoveInPlane.Mode := mcACP6D_MOVE_ABSOLUTE;
			station.Operation.MoveInPlane.Position.X := 0.840;
			station.Operation.MoveInPlane.Position.Y := 0.360;

			station.Commands.MoveInPlane := TRUE;

			IF station.CommandAcknowledge THEN
				station.NextState := TRUE;
			END_IF;
		104:
			station.StateInfo := 'Spin 2';
			// -----------------------------------------------------------------
			station.Operation.Spin.Velocity := -22.0;
			station.Commands.Spin := TRUE;

			IF station.CommandAcknowledge THEN
				station.JumpToState := 199;
			END_IF;
		199:
			station.StateInfo := 'Save macro';
			// -----------------------------------------------------------------
			station.Commands.MacroSave := TRUE;

			IF station.CommandDone THEN
				station.JumpToState := 200;
			END_IF;

		200:
			station.StateInfo := 'Waiting for shuttle to arrive at station';
			// -----------------------------------------------------------------
			station.Loop := 0;

			IF station.NumOccupyingShuttles > 0 THEN
				station.NextState := TRUE;
			END_IF;
		201:
			station.StateInfo := 'Add last arrived shuttle to the station';
			// -----------------------------------------------------------------
			station.Commands.AddShuttle := TRUE;

			IF station.CommandDone THEN
				station.NextState := TRUE;
			END_IF;
		202:
			station.StateInfo := 'Run macro';
			// -----------------------------------------------------------------
			station.Operation.Shuttle := station.Shuttles.List[0];
			station.Commands.MacroRun := TRUE;

			IF station.CommandDone THEN
				station.Loop := station.Loop + 1;
				IF station.Loop < 0 THEN
					station.Commands.MacroRun := FALSE;
				ELSE
					station.JumpToState := 1000;
				END_IF;
			END_IF;
			//		106:
//			station.StateInfo := 'Move to last position';
//			// -----------------------------------------------------------------
//			station.Operation.MoveInPlane.Mode := mcACP6D_MOVE_ABSOLUTE;
//			station.Operation.MoveInPlane.Position.X := 0.840;
//			station.Operation.MoveInPlane.Position.Y := 0.360;
//
//			station.Commands.MoveInPlane := TRUE;
//
//			IF station.CommandAcknowledge THEN
//				station.JumpToState := 199;
//			END_IF;

		1000:
			station.StateInfo := 'Release shuttle to traffic network';
			// -----------------------------------------------------------------
			station.Commands.ReleaseAllShuttles := TRUE;

			IF station.CommandDone THEN
				station.JumpToState := 200;
			END_IF;
	END_CASE;

	// Add macro info for these steps
	IF station.State > 100 AND station.State < 200 THEN
		station.StateInfo := CONCAT('Writing macro - ', station.StateInfo);
	END_IF;

END_ACTION
```

#### station_S3.st
```iecst
ACTION execute_station_S3:
	// Point station reference to this station
	station ACCESS ADR(stations[3]);

	// Station parameters
	station.Station := ADR(S3);
	station.NextStation := ADR(S5);
	station.Parameters.ShuttleCapacity := 1;
	station.Parameters.Zone.BottomLeft.X := 0.720;
	station.Parameters.Zone.BottomLeft.Y := 1.440;
	station.Parameters.Zone.TopRight.X := 0.960;
	station.Parameters.Zone.TopRight.Y := 1.920;

	CASE station.State OF
		0:
			station.StateInfo := 'Activating station';
			// -----------------------------------------------------------------
			IF station.Active THEN
				station.Loop := 0;
				station.JumpToState := 100;
			END_IF;

		100:
			station.StateInfo := 'Movement settings';
			// -----------------------------------------------------------------
			set_movement_parameters_to_default_values;

			station.Operation.Shuttle := station.MacroShuttle;
			station.Operation.MoveArc.EndVelocity := 1.5;
			station.Operation.MoveArc.Angular.Angle := brmPI;
			station.NextState := TRUE;
		101:
			station.StateInfo := 'Move to position 1';
			// -----------------------------------------------------------------
			station.Operation.MoveInPlane.Mode := mcACP6D_MOVE_ABSOLUTE;
			station.Operation.MoveInPlane.Position.X := 0.840;
			station.Operation.MoveInPlane.Position.Y := 1.680;

			station.Commands.MoveInPlane := TRUE;

			IF station.CommandAcknowledge THEN
				station.NextState := TRUE;
			END_IF;
		102:
			station.StateInfo := 'Move figure 8';
			// -----------------------------------------------------------------
			station.Operation.MoveInPlane.Mode := mcACP6D_MOVE_ABSOLUTE;
			station.Operation.MoveArc.Direction := mcACP6D_ARC_COUNTER_CLOCKWISE;
			station.Operation.MoveArc.Angular.Center.X := 0;
			station.Operation.MoveArc.Angular.Center.Y := 0.060;
			station.Commands.MoveArc := TRUE;

			IF station.CommandAcknowledge THEN
				station.NextState := TRUE;
			END_IF;
		103:
			station.StateInfo := 'Move figure 8';
			// -----------------------------------------------------------------
			station.Operation.MoveArc.Direction := mcACP6D_ARC_COUNTER_CLOCKWISE;
			station.Operation.MoveArc.Angular.Center.X := 0;
			station.Operation.MoveArc.Angular.Center.Y := -0.060;
			station.Commands.MoveArc := TRUE;

			IF station.CommandAcknowledge THEN
				station.NextState := TRUE;
			END_IF;
		104:
			station.StateInfo := 'Move figure 8';
			// -----------------------------------------------------------------
			station.Operation.MoveArc.Direction := mcACP6D_ARC_CLOCKWISE;
			station.Operation.MoveArc.Angular.Center.X := 0;
			station.Operation.MoveArc.Angular.Center.Y := -0.060;
			station.Commands.MoveArc := TRUE;

			IF station.CommandAcknowledge THEN
				station.NextState := TRUE;
			END_IF;
		105:
			station.StateInfo := 'Move figure 8';
			// -----------------------------------------------------------------
			station.Operation.MoveArc.Direction := mcACP6D_ARC_CLOCKWISE;
			station.Operation.MoveArc.Angular.Center.X := 0;
			station.Operation.MoveArc.Angular.Center.Y := 0.060;
			station.Commands.MoveArc := TRUE;

			IF station.CommandAcknowledge THEN
				station.NextState := TRUE;
			END_IF;
		106:
			station.StateInfo := 'Check if sequence is complete';
			// -----------------------------------------------------------------
			IF station.Loop < 5 THEN
				station.Loop := station.Loop + 1;
				station.JumpToState := 100;
			ELSE
				station.NextState := TRUE;
			END_IF;
		107:
			station.StateInfo := 'Move to last position';
			// -----------------------------------------------------------------
			station.Operation.MoveArc.Direction := mcACP6D_ARC_COUNTER_CLOCKWISE;
			station.Operation.MoveArc.Angular.Center.X := 0;
			station.Operation.MoveArc.Angular.Center.Y := 0.060;
			station.Operation.MoveArc.EndVelocity := 0;
			station.Commands.MoveArc := TRUE;

			IF station.CommandAcknowledge THEN
				station.JumpToState := 199;
			END_IF;
		199:
			station.StateInfo := 'Save macro';
			// -----------------------------------------------------------------
			station.Commands.MacroSave := TRUE;

			IF station.CommandDone THEN
				station.JumpToState := 200;
			END_IF;

		200:
			station.StateInfo := 'Waiting for shuttle to arrive at station';
			// -----------------------------------------------------------------
			station.Loop := 0;

			IF station.NumOccupyingShuttles > 0 THEN
				station.NextState := TRUE;
			END_IF;
		201:
			station.StateInfo := 'Add last arrived shuttle to the station';
			// -----------------------------------------------------------------
			station.Commands.AddShuttle := TRUE;

			IF station.CommandDone THEN
				station.NextState := TRUE;
			END_IF;
		202:
			station.StateInfo := 'Run macro';
			// -----------------------------------------------------------------
			station.Operation.Shuttle := station.Shuttles.List[0];
			station.Commands.MacroRun := TRUE;

			IF station.CommandDone THEN
				station.JumpToState := 1000;
			END_IF;

		1000:
			station.StateInfo := 'Release shuttle to traffic network';
			// -----------------------------------------------------------------
			station.Commands.ReleaseAllShuttles := TRUE;

			IF station.CommandDone THEN
				station.JumpToState := 200;
			END_IF;
	END_CASE;

	// Add macro info for these steps
	IF station.State > 100 AND station.State < 200 THEN
		station.StateInfo := CONCAT('Writing macro - ', station.StateInfo);
	END_IF;

END_ACTION
```
